{attribute 'enable_dynamic_creation'}
FUNCTION_BLOCK FB_CondiProcessData EXTENDS FB_CondiBase
VAR_INPUT
END_VAR
VAR_OUTPUT
END_VAR
VAR
	eProcDataType : E_ProcDataType;
	iDevice		  : I_Device;
	nCompareValue : DINT;
END_VAR

PROPERTY P_iDevice : I_Device
SET
iDevice := P_iDevice;
END_SET
END_PROPERTY

PROPERTY P_nValue : DINT
SET
nCompareValue := P_nValue;
END_SET
END_PROPERTY

METHOD M_Check : BYTE
VAR_INPUT
	nPreResult : BYTE;
END_VAR

VAR
	bResult			: BOOL;
	nCurrentValue	: DINT;
END_VAR
nCurrentValue := iDevice.M_GetProcData(eProcDataType);

IF eCondition = E_Condition.CONDITION_ProcessVarLEQ THEN
	IF nCurrentValue <= nCompareValue THEN
		bResult := TRUE;
	END_IF
ELSIF eCondition = E_Condition.CONDITION_ProcessVarGEQ THEN
	IF nCurrentValue >= nCompareValue THEN
		bResult := TRUE;
	END_IF	
END_IF

//es wird nur Bit0 entsprechend verknüpft
//Bit1 steht für "Cancel" und wird derzeit nur FB_CondiStepResult verküpft
IF eCondiOperator = E_LogicOperator.LOGIC_OP_AND THEN
	nPreResult.0 := nPreResult.0 AND bResult;
ELSIF eCondiOperator = E_LogicOperator.LOGIC_OP_OR THEN
	nPreResult.0 := nPreResult.0 OR bResult;
END_IF

IF pNextCondi > 0 THEN
	M_Check := pNextCondi^.M_Check(nPreResult);
ELSE
	M_Check  := nPreResult;
END_IF
END_METHOD

PROPERTY P_eProcDataType : E_ProcDataType
SET
eProcDataType := P_eProcDataType;
END_SET
END_PROPERTY

END_FUNCTION_BLOCK

(* stored: Version 1.1.0.1, ProductVersion 3.1.4020.12
   POU FB_CondiProcessData: Id {a418028f-76f1-4526-9fcf-5615a079b25c}, SpecialFunc None
   Property P_iDevice: Id {17c9344d-65ed-42af-879a-8056ac38deb4}
   Set Set: Id {d9c349cc-3ee8-4722-a001-d912904bd897}
   Property P_nValue: Id {69406c7e-ac21-44af-aaab-d84058927e8e}
   Set Set: Id {0909f1df-5a11-4466-be3b-510c83544562}
   Method M_Check: Id {da3bef8f-d630-4fb7-9dd2-08df075fc31f}
   Property P_eProcDataType: Id {f9d3619e-fee1-4fc7-ad5d-31ea4d71b27a}
   Set Set: Id {f9fb3684-c982-4499-a9c7-e6260ba8fe4a} *)
